{attribute addProperty BoxType "EK1122-0000-0018"}
{attribute addProperty Id "Beckhoff_EJx9xxsub_EK1100EK1100_179A0949162"}
{attribute addProperty CRC "97694739"}
{attribute addProperty SizeInBites "16"}
{attribute addProperty SizeInBytes "2"}
TYPE Beckhoff_EJx9xxEK1122_05D2B413 EXTENDS EK1122_179A0949 :
STRUCT
	{attribute addProperty Name "Beckhoff_EJx9xxsub_EK1100"}
	Beckhoff_EJx9xxsub_EK1100 : EK1100_179A0949;
END_STRUCT
END_TYPE

(* stored: Version 1.2.0.0, ProductVersion 3.1.4024.9
   DUT Beckhoff_EJx9xxEK1122_05D2B413: Id {3984aeb0-eadd-43ef-9a73-8cdc5b5cde10} *)
